{attribute 'linkalways'} 
{attribute 'no_explicit_call' := 'This FB is a CLASS and must be accessed using methods or properties'}
{attribute 'enable_dynamic_creation'}
FUNCTION_BLOCK PUBLIC StopCommand EXTENDS AxisCommand
VAR
	_fb : MC_Stop;
	_deceleration : LREAL;
	_jerk : LREAL;
END_VAR

METHOD FB_init : BOOL
VAR_INPUT
	bInitRetains : BOOL; // if TRUE, the retain variables are initialized (warm start / cold start)
	bInCopyCode : BOOL;  // if TRUE, the instance afterwards gets moved into the copy code (online change)
	axis : I_Axis;
END_VAR
_axis := axis;
END_METHOD

METHOD PROTECTED OnExecuting
VAR_INPUT
	stateControl : I_AsyncCommandStateControl;
END_VAR
_fb(
	Axis := _axis._InternalAxisRef,
	Execute := TRUE,
	Deceleration := _deceleration,
	Jerk := _jerk
);

IF _fb.Done THEN
	_fb(Axis := _axis._InternalAxisRef, Execute := FALSE);
	stateControl.Next();
END_IF

IF _fb.CommandAborted THEN
	_fb(Axis := _axis._InternalAxisRef, Execute := FALSE);
	THIS^.Abort();
END_IF

IF _fb.Error THEN
	_fb(Axis := _axis._InternalAxisRef, Execute := FALSE);
	stateControl.Error(_fb.ErrorID);
END_IF
END_METHOD

END_FUNCTION_BLOCK

(* stored: Version 1.1.0.1, ProductVersion 3.1.4024.12
   POU StopCommand: Id {5aedb90c-1a45-4333-8ff4-9287e637597f}, SpecialFunc None
   Folder Constructor: Id {dc0acbb8-17a6-426e-9fbb-199eb0e53e8a}
   Method FB_init: Id {08dabbdf-6250-4037-ba02-16e1df44f728}
   Method OnExecuting: Id {e338eecc-8c22-0d4b-3265-043ee3c3bc83} *)
